Staubli VAL3: CommParameter.dtx

public num port
public string target
public num clients
public num endOfString
public num timeOut
public num baudRate
public string parity
public num bits
public num stopBits
public string mode
public string flowControl
public bool nagle
